// SIMATIC S7-200 project (STEP 7-Micro/WIN), CPU 224 REL 01.11

SYMBOL_TABLE USER1
ON1              I0.0
ON2              I0.1
OFF              I0.2
END_SYMBOL_TABLE

ORGANIZATION_BLOCK MAIN:OB1
TITLE=PROGRAM COMMENTS
BEGIN
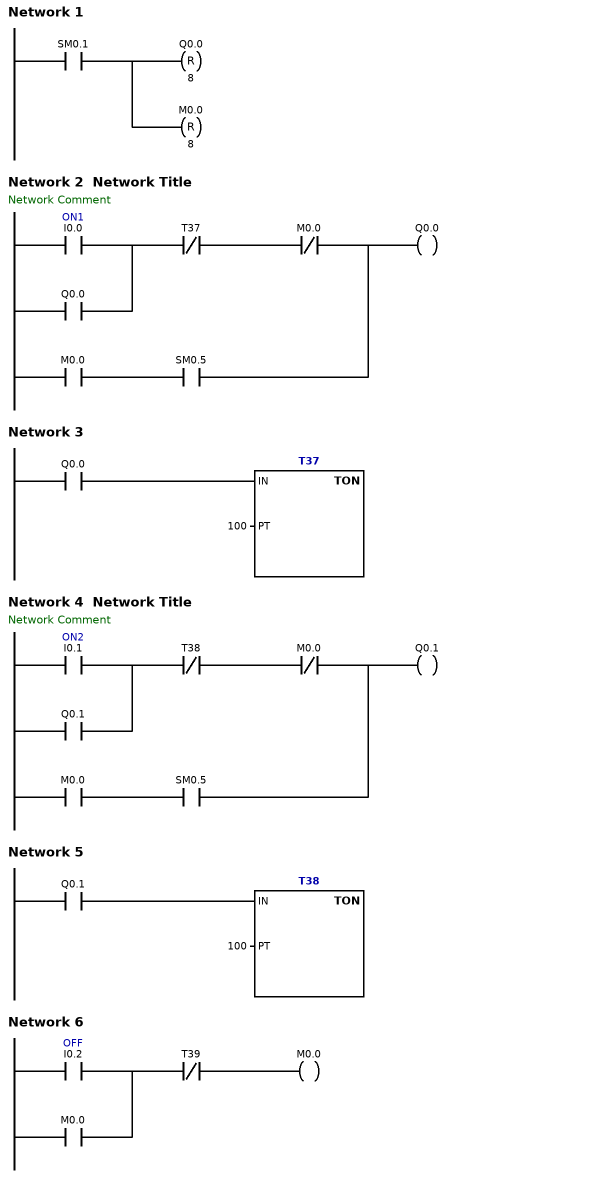
Network 1
LD     SM0.1
R      Q0.0, 8
R      M0.0, 8
Network 2 // Network Title
// Network Comment
LD     ON1:I0.0
O      Q0.0
AN     T37
AN     M0.0
LD     M0.0
A      SM0.5
OLD
=      Q0.0
Network 3
LD     Q0.0
TON    T37, 100
Network 4 // Network Title
// Network Comment
LD     ON2:I0.1
O      Q0.1
AN     T38
AN     M0.0
LD     M0.0
A      SM0.5
OLD
=      Q0.1
Network 5
LD     Q0.1
TON    T38, 100
Network 6
LD     OFF:I0.2
O      M0.0
AN     T39
=      M0.0
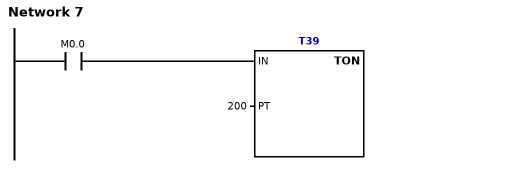
Network 7
LD     M0.0
TON    T39, 200
END_ORGANIZATION_BLOCK
